FUNCTION_BLOCK FB_TestTrigger
VAR_INPUT
    bTestBool : BOOL ;
END_VAR
VAR_OUTPUT
END_VAR
VAR
    rtRisingTrigger : r_trig;
END_VAR

rtRisingTrigger(CLK:=bTestBool);

END_FUNCTION_BLOCK

(* stored: Version 1.1.0.1, ProductVersion 3.1.4022.18
   POU FB_TestTrigger: Id {9c874e7e-d756-4f64-bde6-5fa058895c46}, SpecialFunc None *)
